// TIA Portal project "LearningFactory_4_0_24V_Task02_SensorsSSC_V18" (V18)

(* hardware
DEVICE "ET 200SP-Station_1"  ET 200SP-Station
   slot 0: "Baugruppenträger_0"  Rack  6ES5 710-8MAx1
   slot 1: "PLC"  CPU 1512SP F-1 PN  6ES7 512-1SK01-0AB0  V2.8
      slot 32768: "PROFINET"  X1
   slot 2: "DO1+2"  DQ 16x24VDC/0.5A ST  6ES7 132-6BH01-0BA0  V0.0
      slot 1: "DO1+2"  DQ 16x24VDC/0.5A ST
   slot 3: "DO3+4"  DQ 16x24VDC/0.5A ST  6ES7 132-6BH01-0BA0  V0.0
      slot 1: "DO3+4"  DQ 16x24VDC/0.5A ST
   slot 4: "DO5+6"  DQ 16x24VDC/0.5A ST  6ES7 132-6BH01-0BA0  V0.0
      slot 1: "DO5+6"  DQ 16x24VDC/0.5A ST
   slot 5: "DO7-14"  DQ 4x24VDC/2A HS  6ES7 132-6BD20-0DA0  V2.0
      slot 1: "DO7-14"  DQ 4x24VDC/2A HS
   slot 6: "DO15-22"  DQ 4x24VDC/2A HS  6ES7 132-6BD20-0DA0  V2.0
      slot 1: "DO15-22"  DQ 4x24VDC/2A HS
   slot 7: "DO23-30"  DQ 4x24VDC/2A HS  6ES7 132-6BD20-0DA0  V2.0
      slot 1: "DO23-30"  DQ 4x24VDC/2A HS
   slot 8: "DI1+2"  DI 16x24VDC ST  6ES7 131-6BH01-0BA0  V0.0
      slot 1: "DI1+2"  DI 16x24VDC ST
   slot 9: "DI3+4"  DI 16x24VDC ST  6ES7 131-6BH01-0BA0  V0.0
      slot 1: "DI3+4"  DI 16x24VDC ST
   slot 10: "DI5"  DI 8x24VDC HS  6ES7 131-6BF00-0DA0  V1.0
      slot 1: "DI5"  DI 8x24VDC HS
   slot 11: "DI6"  DI 8x24VDC HS  6ES7 131-6BF00-0DA0  V1.0
      slot 1: "DI6"  DI 8x24VDC HS
   slot 12: "AI7-10"  AI 2xU ST  6ES7 134-6FB00-0BA1  V1.0
      slot 1: "AI7-10"  AI 2xU ST
   slot 13: "End"  Server module  6ES7 193-6PA00-0AA0  V1.1
      slot 1: "End"  Server module
   slot 127: "BA 2xRJ45"  BA 2xRJ45  6ES7 193-6AR00-0AA0  V0.0
      slot 32769: "Port_1"  6ES7 193-6AR00-0AA0
      slot 32770: "Port_2"  6ES7 193-6AR00-0AA0
*)

// ===== PLC "PLC"  CPU 1512SP F-1 PN =====

VAR_GLOBAL   // PLC tag table "SSC - Sensor-Station"
   "QX_SSC_LED_Green_Q5" AT %Q6.4 : Bool;
   "QX_SSC_LED_Yellow_Q6" AT %Q6.5 : Bool;
   "QX_SSC_LED_Red_Q7" AT %Q6.6 : Bool;
   "QX_SSC_LED_Red_Online_Q8" AT %Q6.7 : Bool;
   "IX_SSC_LightBarrierStorage_I3" AT %I4.3 : Bool;
   "IX_SSC_LightBarrierOutsourcing_I4" AT %I4.2 : Bool;
   "IW_SSC_ColorSensor_A1" AT %IW9 : Word;
END_VAR

VAR_GLOBAL   // PLC tag table "Start_Stop"
   "IX_START" AT %I4.4 : Bool;
   "IX_STOP" AT %I4.6 : Bool;
END_VAR

FUNCTION "Task02_ColorSensor" : Void   // FC1, SCL
{ S7_Optimized_Access := 'TRUE' }
VERSION : 0.1
   VAR_INPUT
      Start : Bool;
      ColorSensor : Int;
   END_VAR
   VAR_OUTPUT
      LED_Green : Bool;
      LED_Yellow : Bool;
      LED_Red : Bool;
      LED_Red_Online : Bool;
   END_VAR
BEGIN
   // Program color recognition with LED- display
   // Programm Farberkennung mit Anzeige an LEDs
   // 

   //Pushbutton START
   //Starttaster
   IF #Start THEN
       // Statement section IF


       // Color blue / Farbe blau
       IF #ColorSensor > 17500 AND #ColorSensor < 18500 THEN
           // Statement section IF
           #LED_Green := TRUE;

           // Color White / Farbe weiß
       ELSIF #ColorSensor > 6000 AND #ColorSensor < 7000 THEN
           // Statement section ELSIF
           #LED_Yellow := TRUE;

           // Color red / Farbe rot
       ELSIF #ColorSensor > 14000 AND #ColorSensor < 15000 THEN
           // Statement section ELSIF
           #LED_Red := TRUE;
       ELSE
           // Statement section ELSE
           #LED_Red_Online := TRUE;
       END_IF;


   END_IF;
END_FUNCTION

ORGANIZATION_BLOCK "Main"   // OB1, SCL, ProgramCycle
TITLE = "Main Program Sweep (Cycle)"
{ S7_Optimized_Access := 'TRUE' }
VERSION : 0.1
   VAR_INPUT
      Initial_Call : Bool;   // Initial call of this OB
      Remanence : Bool;   // =True, if remanent data are available
   END_VAR
BEGIN


   // Call subroutine ColorSensor
   // Aufruf Unterprogramm ColorSensor
   "Task02_ColorSensor"(Start:="IX_START",
                        ColorSensor:="IW_SSC_ColorSensor_A1",
                        LED_Green=>"QX_SSC_LED_Green_Q5",
                        LED_Yellow=>"QX_SSC_LED_Yellow_Q6",
                        LED_Red=>"QX_SSC_LED_Red_Q7",
                        LED_Red_Online=>"QX_SSC_LED_Red_Online_Q8");
END_ORGANIZATION_BLOCK